{attribute 'qualified_only'}
{attribute 'strict'}
TYPE SafeState :
(
	Init := 0,
	Close := 1,
	Open := 2,
	CheCkDigit := 3,
	WrongCode := 4
);
END_TYPE

(* stored: Version 1.1.0.1, ProductVersion 3.1.4022.12
   DUT SafeState: Id {02080262-94c0-4c5e-b89f-771bb919f59d} *)
